KUKA KRL data list: A42_rotjoin_global.dat

&ACCESS RV
&COMMENT V_1_4_0
&PARAM DISKPATH = KRC:\R1\BMW_App
&REL 4
DEFDAT A42_rotjoin_global PUBLIC
;********************************
;Date: 07.11.2018
;Programmer: AIUT
;Description: Global positions
;********************************


ENDDAT
